// TwinCAT 3 PLC project GarageNCAxis
// ProgramVersion: 3.1.4024.0
// libraries:
//   CmpBitmapPool, * (System)
//   Tc2_MC2, * (Beckhoff Automation GmbH)
//   Tc2_NC, * (Beckhoff Automation GmbH)
//   Tc2_Standard, * (Beckhoff Automation GmbH)
//   Tc2_System, * (Beckhoff Automation GmbH)
//   Tc3_Module, * (Beckhoff Automation GmbH)
// project tree:
//   / GlobalTextList.TcGTLO, PlcTask.TcTTO (not stored), Visualization Manager.TcVMO (not stored), VISU_TASK.TcTTO
//   POUs/ Blinker.TcPOU, ErrorHandler.TcPOU, GarageDoor.TcPOU, ImagePool.TcIPO (not stored), MAIN.TcPOU, MoveGarageDoor.TcPOU, Visualization.TcVIS
// real-time tasks:
//   TASK PlcTask: cycle T#10ms, priority 20, ADS port 350
//   TASK VISU_TASK: cycle T#200000us, priority 30, ADS port 351
// motion (NC):
//   TASK NC-Task 1 SAF: cycle T#2ms, priority 4, ADS port 501
//   TASK NC-Task 1 SVB: cycle T#10ms, priority 8, ADS port 511
//   AXIS Axis 2 (id 2)
//     General: UnitName=Degree
//     OtherSettings: AllowMotionCmdToSlave=true
//     encoder EncType=19
//       EncPara: ScaleFactorNumerator=0.0054931640625, Offset=2459663.5693, MaxCount=#xffffffff
//     drive DrvType=16
//       DrvPara: MaxCount=#xffffffff, DriveControlDWord=#x00020000
//         Analog: TorqueSetpointScale=10, ScaleFactorActTorque=0.1
//         TimeComp: TaskDelayCycles=1
//     controller CtrType=1
//       CtrPara: PriorControlFactor=1
//         PosDiffControl: Range=20
//         Observer: BandWidth=20
//   AXIS antonio (id 1)
//     General: UnitName=Degree
//     OtherSettings: AllowMotionCmdToSlave=true
//     encoder EncType=19
//       EncPara: ScaleFactorNumerator=0.0054931640625, Offset=-4324197.1783, MaxCount=#xffffffff
//     drive DrvType=16
//       DrvPara: MaxCount=#xffffffff, DriveControlDWord=#x00020000
//         Analog: TorqueSetpointScale=10, ScaleFactorActTorque=0.1
//         TimeComp: TaskDelayCycles=1
//     controller CtrType=1
//       CtrPara: PriorControlFactor=1
//         PosDiffControl: Range=20
//         Observer: BandWidth=20
// I/O:
//   DEVICE Device 3 (EtherCAT) (disabled), AmsNetId 10.0.30.150.4.1
//     Term 1 (EK1100) [EK1100 EtherCAT Coupler (2A E-Bus)]
//       Term 2 (EL1014) [EL1014 4Ch. Dig. Input 24V, 10µs]
//       Term 3 (EL9011) [EL9011 End Terminal]
//   DEVICE Drives (EtherCAT), AmsNetId 10.0.20.83.2.1
//     Drive 4 (Servo 9400 Highline TA CiA 402) [Servo 9400 Highline ECAT V3 TA CiA 402]
//     Drive 6 (Servo 9400 Highline TA CiA 402) [Servo 9400 Highline ECAT V2 TA CiA 402]
// variable links:
//   NC-Task 1 SAF/Axes/Axis 2 <-> Drives (EtherCAT)/Drive 4 (Servo 9400 Highline TA CiA 402)
//     Drive/Inputs/In/nDcOutputTime <-> InfoData/DcOutputShift
//     Drive/Inputs/In/nState1 <-> Cylic Position Mode/Statusword
//     Drive/Inputs/In/nState2 <-> Cylic Position Mode/Statusword @bit 8
//     Drive/Inputs/In/nState4 @bit 1 <-> WcState/InputToggle
//     Drive/Inputs/In/nState4 <-> WcState/WcStateIn
//     Drive/Inputs/In/nState5 <-> Cylic Position Mode/Mode of Operation display
//     Drive/Outputs/Out/nCtrl1 <-> Cylic Position Mode_1/Controlword
//     Drive/Outputs/Out/nCtrl2 <-> Cylic Position Mode_1/Controlword @bit 8
//     Drive/Outputs/Out/nCtrl5 <-> Cylic Position Mode_1/Mode of Operation
//     Drive/Outputs/Out/nDataOut1 <-> Cylic Position Mode_1/Target position
//     Enc/Inputs/In/nDataIn1 <-> Cylic Position Mode/Position actual value (units)
//     Enc/Inputs/In/nDcInputTime <-> InfoData/DcInputShift
//     Enc/Inputs/In/nState4 @bit 1 <-> WcState/InputToggle
//     Enc/Inputs/In/nState4 <-> WcState/WcStateIn
//   NC-Task 1 SAF/Axes/antonio <-> Drives (EtherCAT)/Drive 6 (Servo 9400 Highline TA CiA 402)
//     Drive/Inputs/In/nDcOutputTime <-> InfoData/DcOutputShift
//     Drive/Inputs/In/nState1 <-> Cylic Position Mode/Statusword
//     Drive/Inputs/In/nState2 <-> Cylic Position Mode/Statusword @bit 8
//     Drive/Inputs/In/nState4 @bit 1 <-> WcState/InputToggle
//     Drive/Inputs/In/nState4 <-> WcState/WcStateIn
//     Drive/Inputs/In/nState5 <-> Cylic Position Mode/Mode of Operation display
//     Drive/Outputs/Out/nCtrl1 <-> Cylic Position Mode_1/Controlword
//     Drive/Outputs/Out/nCtrl2 <-> Cylic Position Mode_1/Controlword @bit 8
//     Drive/Outputs/Out/nCtrl5 <-> Cylic Position Mode_1/Mode of Operation
//     Drive/Outputs/Out/nDataOut1 <-> Cylic Position Mode_1/Target position
//     Enc/Inputs/In/nDataIn1 <-> Cylic Position Mode/Position actual value (units)
//     Enc/Inputs/In/nDcInputTime <-> InfoData/DcInputShift
//     Enc/Inputs/In/nState4 @bit 1 <-> WcState/InputToggle
//     Enc/Inputs/In/nState4 <-> WcState/WcStateIn
//   GarageNCAxis/GarageNCAxis Instance <-> Device 3 (EtherCAT)/Term 1 (EK1100)/Term 2 (EL1014)
//     PlcTask Inputs/GarageDoor.bActuationButton <-> Channel 1/Input
//     PlcTask Inputs/GarageDoor.bErrorButton <-> Channel 2/Input
//   GarageNCAxis/GarageNCAxis Instance <-> NC-Task 1 SAF/Axes/Axis 2
//     PlcTask Inputs/GarageDoor.fbMotion.Actuator.NcToPlc <-> Outputs/ToPlc
//     PlcTask Outputs/GarageDoor.fbMotion.Actuator.PlcToNc <-> Inputs/FromPlc
//   GarageNCAxis/GarageNCAxis Instance <-> NC-Task 1 SAF/Axes/antonio
//     PlcTask Inputs/GarageDoor.fbMotion.SecondActuator.NcToPlc <-> Outputs/ToPlc
//     PlcTask Outputs/GarageDoor.fbMotion.SecondActuator.PlcToNc <-> Inputs/FromPlc

CONFIGURATION GarageNCAxis
    RESOURCE PLC ON TwinCAT3
        TASK VISU_TASK(INTERVAL := T#200000us, PRIORITY := 30);
        PROGRAM VisuElems_Visu_Prg WITH VISU_TASK : VisuElems.Visu_Prg;
    END_RESOURCE
END_CONFIGURATION

// ---- POUs/Blinker.TcPOU
FUNCTION_BLOCK Blinker
VAR_INPUT
END_VAR
VAR_OUTPUT
	bBlink : BOOL; //bool variable that sets the light on/off constantly
END_VAR
VAR
	fbTimer1 : TON;
	fbTimer2 : TON;
	fbTimer3 : TON;
	
	iStateFB : INT; //state variable to switch between states in the blinker function block
END_VAR

CASE iStateFB OF
	0:
		bBlink := TRUE;
		fbTimer1.IN := TRUE;
		iStateFB := 10;
	10:	
		IF fbTimer1.Q THEN
			bBlink := FALSE;
			fbTimer1.IN := FALSE;
			fbTimer2.IN := TRUE;
			iStateFB := 20;
		END_IF
	20:
		IF fbTimer2.Q THEN
			bBlink := TRUE;
			fbTimer2.IN := FALSE;
			fbTimer3.IN := TRUE;
			iStateFB := 30;
		END_IF	
	30:
		IF fbTimer3.Q THEN
			bBlink := FALSE;
			fbTimer3.IN := FALSE;
			iStateFB := 0;
		END_IF	
END_CASE

fbTimer1(PT := T#400MS);// timers for blinkers
fbTimer2(PT := T#400MS);
fbTimer3(PT := T#400MS);

END_FUNCTION_BLOCK

// ---- POUs/ErrorHandler.TcPOU
FUNCTION_BLOCK ErrorHandler
VAR_INPUT
	bAxisStatus : BOOL; //checks if the axis has errors
	iInputError : UDINT; //we get the error from the program and handle it here
	bClickedReset : BOOL; //checks whether or not the axis got reset
END_VAR
VAR_OUTPUT
	bEncoderOrPowerError : BOOL; //encoder error or power outage error
	bControllerOr24VError : BOOL; //controller or 24V error
END_VAR
VAR
END_VAR

IF iInputError = 18000 AND bAxisStatus THEN
	bEncoderOrPowerError := TRUE;
	bControllerOr24VError := FALSE;
ELSIF iInputError = 0 AND bAxisStatus THEN
	bEncoderOrPowerError := FALSE;
	bControllerOr24VError := TRUE;
ELSIF iInputError = 0 AND NOT bAxisStatus THEN
	bEncoderOrPowerError := FALSE;
	bControllerOr24VError := FALSE;
END_IF

END_FUNCTION_BLOCK

// ---- POUs/GarageDoor.TcPOU
PROGRAM GarageDoor
VAR
	fbMotion : MoveGarageDoor;
	bActuationButton AT %I* : BOOL; //button that we control through visualization
	bErrorButton AT %I* : BOOL; //button for simulating error
	bDoorOpened : BOOL; //sensor for open door
	bDoorClosed : BOOL; //sensor for close door
	bDoorDriveOverload : BOOL; //sensor for the overload of the door
	bDoorPaused : BOOL; //sensor for pausing the door
	bMotionLight : BOOL; //light that indicates there is motion
	bResetButton : BOOL; //button used to reset the error state
	fPosition : LREAL; //shows the position of the door
	
	bTest1 : BOOL;
	bTest2 : BOOL;
	bTest3 : BOOL;
	
	bTest4 : BOOL;
	bTest5 : BOOL;
	
	bPauseVis : BOOL;
	bErrorVis : BOOL;
	
	bEncOrPwrErr : BOOL; //encoder or power outage error
	bCtrOr24VErr : BOOL; //controller or 24V error
	
	bGearingButton : BOOL;
	
	bAxisMovement : BOOL;
	
	rGearRatio : REAL;
END_VAR

fbMotion.bActuationProgram := bActuationButton;
fbMotion.bError := bErrorButton;
fbMotion.bReset := bResetButton;

bDoorOpened := fbMotion.bOpened;
bDoorClosed := fbMotion.bClosed;
bDoorDriveOverload := fbMotion.bDriveOverload;
bDoorPaused := fbMotion.bPaused;
bMotionLight := fbMotion.bLight;

fPosition := fbMotion.fActPos;

bTest1 := fbMotion.bVis1O;
bTest2 := fbMotion.bVis2O;
bTest3 := fbMotion.bVis3O;

bTest4 := fbMotion.bVis1C;
bTest5 := fbMotion.bVis2C;

bPauseVis := fbMotion.bPauseImg;
bErrorVis := fbMotion.bErrorImg;

bEncOrPwrErr := fbMotion.bEncoderOrPowerErr;
bCtrOr24VErr := fbMotion.bController24VErr;

fbMotion.bGearButton := bGearingButton;

bAxisMovement := fbMotion.bAxisBusy;

fbMotion.rRatioInput := rGearRatio;

fbMotion();

END_PROGRAM

// ---- POUs/MoveGarageDoor.TcPOU
FUNCTION_BLOCK MoveGarageDoor
VAR_INPUT
	bActuationProgram : BOOL; //actuation button for moving the door
	bError : BOOL; //input error
	bReset : BOOL; //reset the axis so it fixes the error
	bGearButton : BOOL; //button that enables the gearing of the axis
	rRatioInput : REAL; //ratio input for the gearing
END_VAR
VAR_OUTPUT
	bClosed : BOOL; //sensor that indicates whether or not the door is closed
	bOpened : BOOL; //sensor that indicates whether or not the door is opened
	bDriveOverload : BOOL; //sensor that indicates whether or not there is an error
	bPaused : BOOL; //sensor that indicates that the door is paused
	bLight : BOOL; //light that shows there is motion
	fActPos : LREAL; //actual position of the axis
	
	bVis1O : BOOL;
	bVis2O : BOOL;
	bVis3O : BOOL;
	bVis1C : BOOL;
	bVis2C : BOOL;
	bErrorImg : BOOL;
	bPauseImg : BOOL;
	
	bEncoderOrPowerErr : BOOL; //all the possible errors
	bController24VErr : BOOL;
	
	bAxisBusy : BOOL; //if the axis is moving dont allow the user to change the gear in/out
END_VAR
VAR
	bInitialActivate : BOOL; //helps set the door to closed at the start
	
	fbActivate : R_TRIG;
	fbInitial : R_TRIG; //helps set the initial value to closed
	fbMsgTrigger : R_TRIG; //helps out with printing the error msg
	
	bActuation : BOOL; //works with the actuation program inside of the function block
	
	iState : UDINT;
	
	Actuator : AXIS_REF; //we refrence the axis
	SecondActuator : AXIS_REF; //we refrence the second axis
	
	McPower : MC_Power; //power and reset function blocks for the axis
	McReset : MC_Reset;
	McMove : MC_MoveAbsolute;
	McStop : MC_Stop;
	
	McPowerSecond : MC_Power; //power and reset function blocks for the axis
	McResetSecond : MC_Reset;
	McMoveSecond : MC_MoveAbsolute;
	McStopSecond : MC_Stop;
	
	McGear : MC_GearIn; 
	McGearDyn : MC_GearInDyn;
	McGearOut : MC_GearOut;
	
	bTempC : BOOL; //helps determine what was the door doing before pause/error
	bTempO : BOOL;
	
	fbError : ErrorHandler;
	
	fbBlinker : Blinker;
	
	iErrorCode : UDINT; //reads the error code that we get so the operator can later resolve the error
	
	sError : STRING(6);
	
	fbInitialGearing : R_TRIG; //sets the initial gearing to off
END_VAR

bInitialActivate := TRUE; //wwe check the state of the door at the start
fbInitial(CLK := TRUE);
IF fbInitial.Q THEN
	bClosed := TRUE; //we have set the door to closed at the start (only activates the first time we run the program
END_IF


CASE iState OF
	0:	
		IF McPower.Enable THEN
			iState := 10;
		END_IF
		
	5: //turning actuation off
		bActuation := FALSE;
		iState := 0; //return to the first state
		
	10:
		fbActivate(CLK := bActuationProgram);
		IF fbActivate.Q THEN
			bActuation := TRUE;
		END_IF
		bTempO := FALSE;
		bTempC := FALSE;
		IF bActuation THEN
			iState := 20; //if we click the button go to the next state and check it's state
		END_IF
		
	15:
		bActuation := FALSE;
		iState := 100;	
		
	20:
		IF bClosed THEN
			iState := 40; //open state
		ELSIF bOpened THEN
			iState := 50; //close state
		ELSE
			iState := 999;// driveoverload state
		END_IF
		
	30:
		bActuation := FALSE;
		iState := 999;
		
	40: //the door is closed we open it
		fbMsgTrigger(CLK := FALSE);
		
		bClosed := FALSE;	
		IF bActuation THEN
			bLight := TRUE;
			bTempO := TRUE;
			McMove(Axis := Actuator, //we open the door (100 means openned)
					Position := 180,
					Velocity := 70,
					Acceleration := 100,
					Deceleration := 100,
					Jerk := 100000,
					Execute := TRUE);
			iState := 45;	
		END_IF
		
	45:	//check if the movement is done
		fbActivate(CLK := bActuationProgram); //incase we want to pause it
		IF fbActivate.Q THEN
			bActuation := FALSE;
		END_IF
		IF bError OR McMove.Error THEN
			iState := 30; //incase the door goes to error
		END_IF
		IF bActuation THEN	
			IF McMove.Done AND NOT McMove.Error THEN
				McMove(Axis := Actuator,Execute := FALSE); //we turn it off
				bOpened := TRUE;
				bLight := FALSE;
				iState := 5;
			END_IF
		ELSE
			bPaused := TRUE;
			iState := 15;	
		END_IF
		
	50: //door is opened we close it
		fbMsgTrigger(CLK := FALSE);
	
		bOpened := FALSE;	
		IF bActuation THEN
			bLight := TRUE;
			bTempC := TRUE;
			McMove(Axis := Actuator, //we close the door  (0 means openned)
					Position := 0,
					Velocity := 70,
					Acceleration := 100,
					Deceleration := 100,
					Jerk := 100000,
					Execute := TRUE);
			iState := 55; //check if the movement is done
		END_IF
		
	55: //check if the movement is done
		fbActivate(CLK := bActuationProgram); //incase we want to pause it
		IF fbActivate.Q THEN
			bActuation := FALSE;
		END_IF
		IF bError OR McMove.Error THEN
			iState := 30; //incase the door goes to error
		END_IF
		IF bActuation THEN
			
	
			IF McMove.Done AND NOT McMove.Error THEN
				McMove(Axis := Actuator,Execute := FALSE); //we turn it off
				bClosed := TRUE;
				bLight := FALSE;
				iState := 5;
			END_IF
		ELSE
			bPaused := TRUE;
			iState := 15;	
		END_IF
		
	100: //pause state
		//bVis1O := FALSE;
		//bVis2O := FALSE;
		//bVis3O := FALSE;
		//bVis1C := FALSE;
		//bVis2C := FALSE;
		//bPauseImg := TRUE;
		
		bLight := FALSE;
		fbActivate(CLK := bActuationProgram);		
		IF fbActivate.Q THEN
			bActuation := TRUE;
			bPaused := FALSE; //we turn off the pause light
		END_IF
		McStop(Axis := Actuator,
				Deceleration := 300,
				Execute := TRUE);
		IF bActuation AND bTempC THEN
			bLight := TRUE;
			bTempC := FALSE;
			McStop(Axis := Actuator,Execute := FALSE);
			McMove(Axis := Actuator,Execute := FALSE);
			iState := 40;
		ELSIF bActuation AND bTempO THEN
			bLight := TRUE;
			bTempO := FALSE;
			McStop(Axis := Actuator,Execute := FALSE);
			McMove(Axis := Actuator,Execute := FALSE);
			iState := 50;	
		END_IF
		
	999: //error state	
		bErrorImg := TRUE;
		fbMsgTrigger(CLK := TRUE);
		IF fbMsgTrigger.Q THEN
			ADSLOGSTR(msgCtrlMask := ADSLOG_MSGTYPE_ERROR OR ADSLOG_MSGTYPE_MSGBOX,
				msgFmtStr := 'Error ID: %s',
				strArg := sError);
		END_IF

		McReset(Axis := Actuator,Execute := bReset); //resets the axis after the error has been resolved
		
		bLight := fbBlinker.bBlink;
		fbBlinker();
		bDriveOverload := TRUE;
		fbActivate(CLK := bActuationProgram);		
		IF fbActivate.Q THEN
			bActuation := TRUE;
			bPaused := FALSE; //we turn off the pause light
		END_IF
		McStop(Axis := Actuator,
				Deceleration := 300,
				Execute := TRUE);
		IF bActuation AND bTempC THEN
			bErrorImg := FALSE;
			bDriveOverload := FALSE;
			bLight := TRUE;
			bTempC := FALSE;
			McStop(Axis := Actuator,Execute := FALSE);
			McMove(Axis := Actuator,Execute := FALSE);
			iState := 40;
		ELSIF bActuation AND bTempO THEN
			bErrorImg := FALSE;
			bDriveOverload := FALSE;
			bLight := TRUE;
			bTempO := FALSE;
			McStop(Axis := Actuator,Execute := FALSE);
			McMove(Axis := Actuator,Execute := FALSE);
			iState := 50;	
		END_IF
		
END_CASE 
Actuator.ReadStatus(); //referencing the axis to the function blocks
SecondActuator.ReadStatus();
McPower(Axis := Actuator,Enable := TRUE,Enable_Positive := TRUE,Enable_Negative := TRUE);
McPowerSecond(Axis := SecondActuator,Enable := TRUE,Enable_Positive := TRUE,Enable_Negative := TRUE);
McReset(Axis := Actuator);
McMove(Axis := Actuator);
McStop(Axis := Actuator);
McResetSecond(Axis := SecondActuator);
McMoveSecond(Axis := SecondActuator);
McStopSecond(Axis := SecondActuator);
SecondActuator.ReadStatus();
fActPos := Actuator.NcToPlc.ActPos;
iErrorCode := Actuator.NcToPlc.ErrorCode;

fbError.iInputError := iErrorCode;
fbError.bAxisStatus := McMove.Error;
bEncoderOrPowerErr := fbError.bEncoderOrPowerError;
bController24VErr := fbError.bControllerOr24VError;
fbError();

sError := TO_STRING(iErrorCode);
// ***Gearing the 2 axis***
IF NOT McMove.Busy THEN
	McGearDyn(Master := Actuator,
				Slave := SecondActuator,
				GearRatio := rRatioInput,
				Enable := NOT bGearButton);
	McGearOut(Slave := SecondActuator,Execute := bGearButton);
END_IF
////******////

bAxisBusy := McMove.Busy;

IF bTempO THEN
	//bErrorImg := FALSE;
	//bPauseImg := FALSE;
	bVis1C := FALSE;
	bVis2C := FALSE;
	IF fActPos > 50.0 THEN
		bVis1O := TRUE;
	END_IF
	IF fActPos > 100.0 THEN
		bVis2O := TRUE;
		bVis1O := FALSE;
	END_IF
	IF fActPos > 150.0 THEN
		bVis2O := FALSE;
		bVis3O := TRUE;
	END_IF
END_IF

IF bTempC THEN
	//bErrorImg := FALSE;
	//bPauseImg := FALSE;
	bVis1O := FALSE;
	bVis2O := FALSE;
	IF fActPos < 150.0 THEN
		bVis1C := TRUE;
		bVis3O := FALSE;
	END_IF
	IF fActPos < 100.0 THEN
		bVis2C := TRUE;
		bVis1C := FALSE;
	END_IF
	IF fActPos < 50.0 THEN
		bVis2C := FALSE;
	END_IF
END_IF

END_FUNCTION_BLOCK

// ---- POUs/MAIN.TcPOU
PROGRAM MAIN
VAR
END_VAR

GarageDoor();

END_PROGRAM

// ---- GlobalTextList.TcGTLO
TEXTLIST GlobalTextList
  219 = '%f'
  90 = '%i'
  509 = '%r'
  596 = 'Actuation'
  448 = 'Actuator position'
  818 = 'Axis Position'
  961 = 'Closed'
  917 = 'Drive Overload'
  130 = 'Gear IN'
  709 = 'Gear OUT'
  534 = 'hi'
  5 = 'Opened'
  837 = 'Paused'
  184 = 'Reset Axis'
  739 = 'sda'
  345 = 'Simulate Error'
  608 = 'There seems to be an error. Please check if the controller is turned on and make sure that the 24V switch is turned on. After that make sure to reset the axis.'
  819 = 'There seems to be an error. Please check if the encoder is connected properly and make sure that the power is turned on.'
  395 = 'There seems to be an error. Please check if the encoder is connected properly and make sure that the power is turned on. After that make sure to reset the axis.'
  782 = 'There seems to be an error. Please check if the resolver is connected properly and make sure that the power is turned on. After that make sure to reset  the axis. If everything seems fine just reset the axis.'
  882 = 'There seems to be an error. Please check if the resolver is connected properly and make sure that the power is turned on. After that make sure to reset the axis.'
END_TEXTLIST

// ---- POUs/Visualization.TcVIS
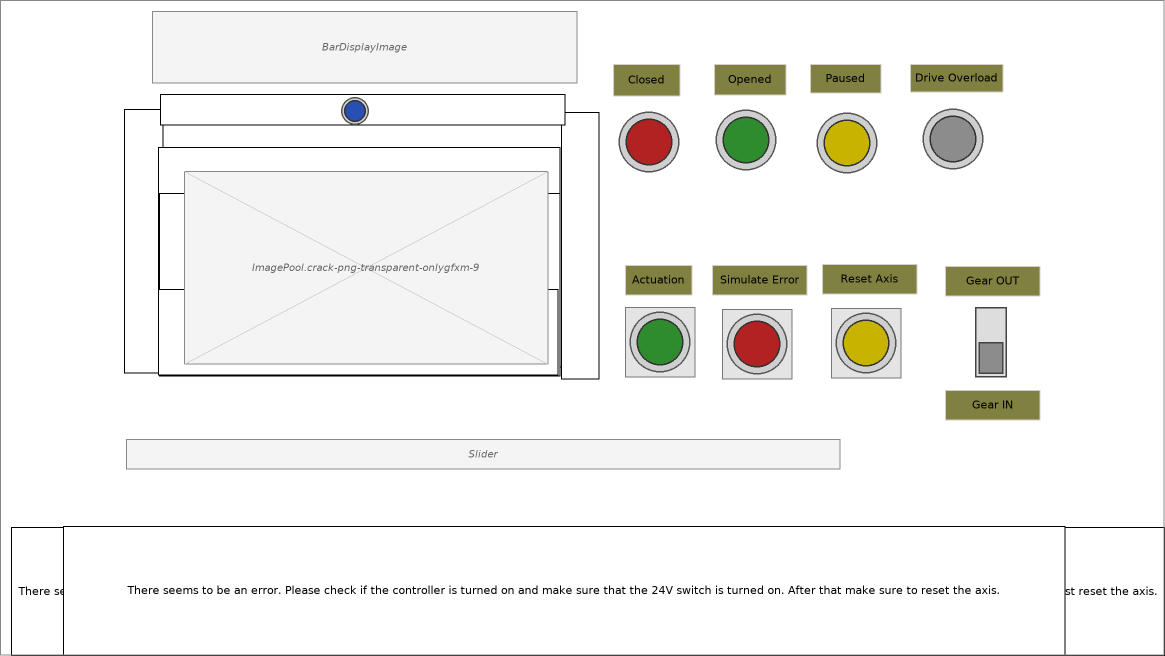
VISUALIZATION Visualization  // 1165x656
    Rectangle (161,123 402x244)
    Rectangle (124,109 39x264)
    Rectangle (561,112 38x267)
    Rectangle (160,94 405x31)
    Lamp1 (339,92 32x38), variable: GarageDoor.bMotionLight, style: Lamp-Lamp1-Blue
    Lamp1 (614,107 70x70), variable: GarageDoor.bDoorClosed, style: Lamp-Lamp1-Red
    Lamp1 (711,105 70x70), variable: GarageDoor.bDoorOpened, style: Lamp-Lamp1-Green
    Lamp1 (812,108 70x70), variable: GarageDoor.bDoorPaused, style: Lamp-Lamp1-Yellow
    Lamp1 (918,104 70x70), variable: GarageDoor.bDoorDriveOverload, style: Lamp-Lamp1-Gray
    PushSwitch (625,307 70x70), variable: GarageDoor.bActuationButton, behaviour: TAP, style: Switch-PushSwitch-Green
    PushSwitch (722,309 70x70), variable: GarageDoor.bErrorButton, behaviour: TAP, style: Switch-PushSwitch-Red
    Rectangle (161,274 399x96), invisible if: NOT GarageDoor.bTest1
    Rectangle (158,147 402x225), invisible if: NOT GarageDoor.bTest3
    Rectangle (160,205 399x166), invisible if: NOT GarageDoor.bTest2
    Rectangle (159,193 401x183), invisible if: NOT GarageDoor.bTest4
    Rectangle (158,289 400x86), invisible if: NOT GarageDoor.bTest5
    Image (184,171 364x193), invisible if: NOT GarageDoor.bErrorVis, image: ImagePool.crack-png-transparent-onlygfxm-9
    Textfield (613,64 67x32), "Closed", colour toggle: GarageDoor.bDoorClosed
    Textfield (714,64 72x31), "Opened", colour toggle: GarageDoor.bDoorOpened
    Textfield (810,64 71x29), "Paused", colour toggle: GarageDoor.bDoorPaused
    Textfield (910,64 93x28), "Drive Overload", colour toggle: GarageDoor.bDoorDriveOverload
    Textfield (625,265 67x30), "Actuation", colour toggle: GarageDoor.bActuationButton
    Textfield (712,265 95x30), "Simulate Error", colour toggle: GarageDoor.bErrorButton
    BarDisplayImage (152,11 425x72), value: GarageDoor.fPosition, style: BarDisplayImage-Gray, scale format: %.1f, scale 0..180
        p518627256: Axis Position
    PushSwitch (831,308 70x70), variable: GarageDoor.bResetButton, behaviour: TAP, style: Switch-PushSwitch-Yellow
    Textfield (822,264 95x30), "Reset Axis", colour toggle: GarageDoor.bErrorButton
    Rectangle (11,527 1154x129), "There seems to be an error. Please check if the resolver is connected properly and make sure that the power is turned on. After that make sure to reset the axis. If everything seems fine just reset the axis.", invisible if: NOT GarageDoor.bEncOrPwrErr
    Rectangle (63,526 1002x129), "There seems to be an error. Please check if the controller is turned on and make sure that the 24V switch is turned on. After that make sure to reset the axis.", invisible if: NOT GarageDoor.bCtrOr24VErr
    DipSwitch (956,307 70x70), variable: GarageDoor.bGearingButton, input disabled if: GarageDoor.bAxisMovement, behaviour: TOGGLE, style: Switch-DipSwitch-Gray
    Textfield (945,266 95x30), "Gear OUT", colour toggle: GarageDoor.bGearingButton
    Textfield (945,390 95x30), "Gear IN", colour toggle: NOT GarageDoor.bGearingButton
    Slider (126,439 714x30), variable: GarageDoor.rGearRatio, input disabled if: GarageDoor.bAxisMovement, scale 0..2
END_VISUALIZATION
